--- Backups/Controller2/RAPID/TASK1/PROGMOD/CalibData.mod ---
MODULE CalibData
    PERS tooldata Tool_cow_catcher:=[TRUE,[[0,35.982,200],[1,0,0,0]],[1,[0,0,1],[1,0,0,0],0,0,0]];
    PERS tooldata Tool_Stack:=[TRUE,[[0,50,519.006],[1,0,0,0]],[1,[0,0,1],[1,0,0,0],0,0,0]];
    TASK PERS wobjdata wokOb_stak:=[FALSE,TRUE,"",[[1085.231623935,1226.713832798,-131.071212416],[0.707106781,0,0,-0.707106781]],[[0,0,0],[1,0,0,0]]];
    TASK PERS wobjdata WokOb_feed:=[FALSE,TRUE,"",[[1185.402623935,-706.018167202,-184.071212416],[0,1,0,0]],[[0,0,0],[1,0,0,0]]];
    TASK PERS wobjdata WokOb_feed1:=[FALSE,TRUE,"",[[1185.402623935,-706.018167202,-184.071212416],[0,1,0,0]],[[0,0,0],[1,0,0,0]]];
    TASK PERS wobjdata WokOb_Train_Top:=[FALSE,TRUE,"",[[58.90254417,-81.246884277,-27.346593322],[1,0.000000015,-0.00000002,-0.000000114]],[[-437.993,1154.838,527.576],[0,0,0.87019971,0.492699163]]];
    TASK PERS wobjdata WokOb_tarin_Front:=[FALSE,TRUE,"",[[58.90254417,-81.246884277,-27.346593322],[1,0.000000015,-0.00000002,-0.000000114]],[[-387.993,1035.72,66.547],[0.509717505,0.490089854,0.490089854,0.509717505]]];
    TASK PERS wobjdata Stand_tool_3:=[FALSE,TRUE,"",[[-537.392313736,-1111.43668764,-49.051212721],[0.707183689,0.000000377,0.000000377,-0.707029865]],[[0,0,0],[1,0,0,0]]];
    PERS tooldata Tooldata_2:=[TRUE,[[0,50,519.006],[1,0,0,0]],[1,[0,0,1],[1,0,0,0],0,0,0]];
    PERS tooldata Tooldata_3:=[TRUE,[[0,35.982,200],[1,0,0,0]],[1,[0,0,1],[1,0,0,0],0,0,0]];
    TASK PERS wobjdata WokOb_feed_1_Caw:=[FALSE,TRUE,"",[[1151.349623935,525.320832798,-184.071212416],[0,1,0,0]],[[0,0,0],[1,0,0,0]]];
    TASK PERS wobjdata WorOb_Stacl_Rb3:=[FALSE,TRUE,"",[[1166.594351677,998.920009045,-48.014532261],[0.705216396,-0.025578864,-0.025682184,-0.708064956]],[[0,0,0],[1,0,0,0]]];
ENDMODULE

--- Backups/Controller2/RAPID/TASK1/PROGMOD/Module1.mod ---
MODULE Module1
        CONST robtarget Target_10:=[[221.184118017,1602.844398512,1266.446017213],[0.128764321,-0.327741314,0.934862358,0.045141464],[-1,0,-1,0],[9E+09,9E+09,9E+09,9E+09,9E+09,9E+09]];
    CONST robtarget Target_20:=[[370.000026729,589.040405274,551.077515218],[0.04939984,-0.01732251,0.998628486,0.000856886],[-1,0,-1,0],[9E+09,9E+09,9E+09,9E+09,9E+09,9E+09]];
    CONST robtarget Target_30_up:=[[414.854817462,671.346228764,341.000522266],[0.000000533,0.00010877,0.999999994,0],[-1,0,0,0],[9E+09,9E+09,9E+09,9E+09,9E+09,9E+09]];
    CONST robtarget Target_30:=[[414.855137357,671.346228729,41.000522266],[0.000000533,0.00010877,0.999999994,0],[-1,0,0,0],[9E+09,9E+09,9E+09,9E+09,9E+09,9E+09]];
    CONST robtarget Target_40:=[[635.144122191,584.664958178,1616.637616509],[0.169784564,-0.794718952,0.515233089,0.27226798],[0,0,-1,0],[9E+09,9E+09,9E+09,9E+09,9E+09,9E+09]];
    CONST robtarget Target_50:=[[566.954133975,747.917817416,1065.318925343],[0.043909951,-0.83413114,0.542350178,0.090296418],[0,0,-1,0],[9E+09,9E+09,9E+09,9E+09,9E+09,9E+09]];
    CONST robtarget Target_60:=[[348.821647049,691.581522758,639.450946441],[0,-0.707106781,0.707106781,0],[0,0,0,0],[9E+09,9E+09,9E+09,9E+09,9E+09,9E+09]];
    CONST robtarget Target_70:=[[172.450821148,1938.736452761,-61.688697976],[0.659237738,-0.298307072,-0.108561129,-0.681639917],[1,0,-1,0],[9E+09,9E+09,9E+09,9E+09,9E+09,9E+09]];
    CONST robtarget Target_80:=[[569.616153696,1591.274414834,107.994145107],[0.624643546,-0.339078797,-0.046011146,-0.701946568],[1,-1,0,0],[9E+09,9E+09,9E+09,9E+09,9E+09,9E+09]];
    CONST robtarget Target_90:=[[387.500477242,662.643098431,-11.713507029],[0.624643546,-0.339078797,-0.046011146,-0.701946568],[1,0,-1,0],[9E+09,9E+09,9E+09,9E+09,9E+09,9E+09]];
    CONST robtarget Target_110:=[[166.316566086,558.37413423,-395.581097695],[0.714499458,0.106310973,-0.106526851,-0.683257295],[0,0,1,0],[9E+09,9E+09,9E+09,9E+09,9E+09,9E+09]];
    CONST robtarget Target_120:=[[-187.554461139,446.991796248,-213.907700592],[0.722131676,-0.014348091,0.019578353,-0.691329634],[0,0,1,0],[9E+09,9E+09,9E+09,9E+09,9E+09,9E+09]];
    CONST robtarget Target_140:=[[439.260504662,249.044211181,306.866921641],[0.012111654,0.04598783,0.712802443,-0.699750744],[1,-1,0,0],[9E+09,9E+09,9E+09,9E+09,9E+09,9E+09]];
    CONST robtarget Target_170:=[[536.884549621,570.585995165,-1132.877964218],[0.000000105,0.349155725,-0.000000008,0.937064715],[-1,0,-1,0],[9E+09,9E+09,9E+09,9E+09,9E+09,9E+09]];
    CONST robtarget Target_150:=[[205.16784185,570.586,-521.43503171],[-0.000000103,0.147809407,0.000000016,0.989015864],[0,-1,0,0],[9E+09,9E+09,9E+09,9E+09,9E+09,9E+09]];
    CONST robtarget Target_160:=[[178.331522758,542.515647049,-380.296079672],[0,0,0,1],[0,0,0,0],[9E+09,9E+09,9E+09,9E+09,9E+09,9E+09]];
    CONST robtarget Target_180:=[[416.962146713,864.683571188,1161.560654219],[0.40242565,-0.070024337,0.596108152,-0.691234591],[0,0,-1,0],[9E+09,9E+09,9E+09,9E+09,9E+09,9E+09]];
    CONST robtarget Target_190:=[[602.180688228,288.578411913,1239.026266106],[0.132681117,0.091945772,0.703686394,-0.691930022],[0,0,-1,0],[9E+09,9E+09,9E+09,9E+09,9E+09,9E+09]];
    CONST robtarget Target_Ro3_Cow_Pre_Last:=[[414.854817462,671.346228764,341.000522267],[0.000000533,0.00010877,0.999999994,0],[-1,0,0,0],[9E+09,9E+09,9E+09,9E+09,9E+09,9E+09]];
    CONST robtarget Target_Ro3_Cow_Last:=[[414.855137357,671.346228729,41.000522267],[0.000000533,0.00010877,0.999999994,0],[-1,0,0,0],[9E+09,9E+09,9E+09,9E+09,9E+09,9E+09]];
    CONST robtarget Target_R3_Caw_Pre_Last:=[[198.331522758,542.515647049,-580.296079672],[0.706823316,0.020019999,-0.020019999,-0.706823316],[-1,-1,0,0],[9E+09,9E+09,9E+09,9E+09,9E+09,9E+09]];
    CONST robtarget Target_200:=[[537.449802278,525.320832798,-1349.697350072],[0,0.093718973,0,0.995598691],[-1,0,-1,0],[9E+09,9E+09,9E+09,9E+09,9E+09,9E+09]];
    CONST robtarget Target_210:=[[395.399205293,525.320832798,-1001.535802608],[0.706823316,0.020019999,-0.020019999,-0.706823316],[-1,-1,0,0],[9E+09,9E+09,9E+09,9E+09,9E+09,9E+09]];
    CONST robtarget Target_R3_Caw_Last:=[[198.331522758,542.515647049,-380.296079672],[0.706823316,0.020019999,-0.020019999,-0.706823316],[-1,-1,0,0],[9E+09,9E+09,9E+09,9E+09,9E+09,9E+09]];
    CONST robtarget Target_R3_Caw_aT_Pre_Last:=[[602.180688228,308.563002126,1239.811220903],[0.132681117,0.091945772,0.703686394,-0.691930022],[0,0,-1,0],[9E+09,9E+09,9E+09,9E+09,9E+09,9E+09]];
    CONST robtarget Target_R3_Caw_aT_Last:=[[439.260504662,269.028801394,307.651876438],[0.009281573,0.046641452,0.754191684,-0.65493002],[0,0,-1,0],[9E+09,9E+09,9E+09,9E+09,9E+09,9E+09]];
    CONST robtarget Target_230:=[[431.630872596,635.901601801,1236.076927583],[0.024057172,-0.814914042,0.571422358,0.093876759],[0,0,-1,0],[9E+09,9E+09,9E+09,9E+09,9E+09,9E+09]];
    CONST robtarget Target_Ro3_Stack_Pre_last:=[[242.865175793,579.269518535,748.277875669],[0.025682184,0.708064956,-0.705216396,-0.025578864],[0,0,0,0],[9E+09,9E+09,9E+09,9E+09,9E+09,9E+09]];
    CONST robtarget Target_Ro3_Stack_last:=[[228.375978011,579.211110467,548.803416812],[0.025682184,0.708064956,-0.705216396,-0.025578864],[0,0,0,0],[9E+09,9E+09,9E+09,9E+09,9E+09,9E+09]];
    CONST robtarget Target_220:=[[578.676966526,497.743647902,1659.839754198],[0.150831029,-0.765727927,0.566419369,0.264725973],[0,0,-1,0],[9E+09,9E+09,9E+09,9E+09,9E+09,9E+09]];
    CONST robtarget Target_240:=[[49.842979194,487.554033752,-1340.183033329],[0.336292984,-0.171245379,-0.062328221,-0.923957381],[-1,0,-1,0],[9E+09,9E+09,9E+09,9E+09,9E+09,9E+09]];
    CONST robtarget Target_250:=[[283.995850065,381.102635573,-1044.400341171],[0.707106781,0,0,-0.707106781],[-1,-1,1,0],[9E+09,9E+09,9E+09,9E+09,9E+09,9E+09]];
    CONST robtarget Target_Rb3_Stack_Pre_Last:=[[270.393522758,498.685647049,-819.068079672],[0.707106781,0,0,-0.707106781],[-1,0,0,0],[9E+09,9E+09,9E+09,9E+09,9E+09,9E+09]];
    CONST robtarget Target_Rb3_Stack_Last:=[[270.393522758,498.685647049,-299.068079672],[0.707106781,0,0,-0.707106781],[-1,0,0,0],[9E+09,9E+09,9E+09,9E+09,9E+09,9E+09]];
    CONST robtarget Target_Stack_2_Pre:=[[168.638525927,1312.987191107,-158.731374197],[0.924786368,-0.310928816,0.214202621,-0.047017889],[1,1,-2,0],[9E+09,9E+09,9E+09,9E+09,9E+09,9E+09]];
    CONST robtarget Target_Stack_4_last:=[[389.005720296,705.812701337,80.121150632],[0.961548171,-0.165322925,0.204449569,-0.07933359],[1,-1,0,0],[9E+09,9E+09,9E+09,9E+09,9E+09,9E+09]];
    CONST robtarget Target_Stack_3_Pre_last:=[[389.005720296,877.311368754,-22.777863329],[0.623819913,-0.261468638,0.027666715,-0.736014552],[1,-1,0,0],[9E+09,9E+09,9E+09,9E+09,9E+09,9E+09]];
    CONST robtarget Target_Stack_1_Start:=[[-788.497531681,1603.313448753,-159.059404418],[0.940109898,-0.316080846,-0.12465014,0.027360947],[0,1,-1,0],[9E+09,9E+09,9E+09,9E+09,9E+09,9E+09]];
    CONST robtarget Target_Stack_3_last:=[[389.005720296,963.060702463,-74.227370309],[0.961548171,-0.165322925,0.204449569,-0.07933359],[1,-1,0,0],[9E+09,9E+09,9E+09,9E+09,9E+09,9E+09]];
    CONST robtarget Target_270:=[[381.16653399,952.850551141,-196.906188778],[0.952856429,-0.264493422,0.136128666,-0.059806695],[1,0,-1,0],[9E+09,9E+09,9E+09,9E+09,9E+09,9E+09]];
    CONST robtarget Target_270_2:=[[381.16652599,1124.349221645,-299.805197594],[0.952856429,-0.264493422,0.136128666,-0.059806695],[1,1,-1,0],[9E+09,9E+09,9E+09,9E+09,9E+09,9E+09]];
!***********************************************************
    !
    ! Module:  Module1
    !
    ! Description:
    !   <Insert description here>
    !
    ! Author: haba0028
    !
    ! Version: 1.0
    !
    !***********************************************************


    !***********************************************************
    !
    ! Procedure main
    !
    !   This is the entry point of your program
    !
    !***********************************************************
    PROC main()
        !Add your code here
        SetDo doAt_Tool_SC1,0;
        SetDO doGrepCaw,0;
        SetDo doGrepStak,0;
        WaitDI di_Atctive,1;





        Path_Att_tool_cow;
        Path_Att_cow_tR;
        Path_Att_cow_tT;
        Path_diAtt_tool_cow;


        Path_Rob3_att_tool_stak;
        Path_Rb3_Att_Stack_tR;
        Path_Rob3_att_tT_Stack;
        Path_Rob3_diatt_tool_stak;



!        Path_Rob3_att_tT_Stack;
    ENDPROC

    PROC Path_Att_tool_cow()
        MoveJ Target_10,v1000,fine,tool0\WObj:=Stand_tool_3;
        MoveL Target_20,v1000,fine,tool0\WObj:=Stand_tool_3;
        MoveL Target_Ro3_Cow_Pre_Last,v1000,fine,tool0\WObj:=Stand_tool_3;
        MoveL Target_Ro3_Cow_Last,v1000,fine,tool0\WObj:=Stand_tool_3;
        WaitTime 0.3;
        SetDo doAt_Tool_SC1,1;
        WaitTime 1;
        MoveL Target_Ro3_Cow_Pre_Last,v1000,fine,Tool_cow_catcher\WObj:=Stand_tool_3;
        MoveL Target_20,v1000,fine,Tool_cow_catcher\WObj:=Stand_tool_3;
        MoveL Target_10,v1000,fine,Tool_cow_catcher\WObj:=Stand_tool_3;
    ENDPROC
    PROC Path_diAtt_tool_cow()
        WaitTime 0.3;
        MoveJ Target_10,v1000,fine,Tool_cow_catcher\WObj:=Stand_tool_3;
        MoveL Target_20,v1000,fine,Tool_cow_catcher\WObj:=Stand_tool_3;
        MoveL Target_Ro3_Cow_Pre_Last,v1000,fine,Tool_cow_catcher\WObj:=Stand_tool_3;
        MoveL Target_Ro3_Cow_Last,v1000,fine,tool0\WObj:=Stand_tool_3;
        WaitTime 0.3;
        SetDo doAt_Tool_SC1,0;
        WaitTime 1;
        MoveL Target_Ro3_Cow_Pre_Last,v1000,fine,tool0\WObj:=Stand_tool_3;
        MoveL Target_20,v1000,fine,tool0\WObj:=Stand_tool_3;
        MoveL Target_10,v1000,fine,tool0\WObj:=Stand_tool_3;
    ENDPROC

    PROC Path_Rob3_att_tool_stak()
        MoveJ Target_220,v1000,fine,tool0\WObj:=WorOb_Stacl_Rb3;
        MoveL Target_230,v1000,fine,tool0\WObj:=WorOb_Stacl_Rb3;
        MoveL Target_Ro3_Stack_Pre_last,v1000,fine,tool0\WObj:=WorOb_Stacl_Rb3;
        MoveL Target_Ro3_Stack_last,v1000,fine,tool0\WObj:=WorOb_Stacl_Rb3;
        WaitTime 0.3;
        SetDo doAt_Tool_SC1,1;
        WaitTime 1;
        MoveL Target_Ro3_Stack_Pre_last,v1000,fine,Tool_Stack\WObj:=WorOb_Stacl_Rb3;
        MoveL Target_230,v1000,fine,Tool_Stack\WObj:=WorOb_Stacl_Rb3;
        MoveL Target_220,v1000,fine,Tool_Stack\WObj:=WorOb_Stacl_Rb3;
    ENDPROC

    PROC Path_Rob3_diatt_tool_stak()
        MoveJ Target_220,v1000,fine,Tool_Stack\WObj:=WorOb_Stacl_Rb3;
        MoveL Target_230,v1000,fine,Tool_Stack\WObj:=WorOb_Stacl_Rb3;
        MoveL Target_Ro3_Stack_Pre_last,v1000,fine,Tool_Stack\WObj:=WorOb_Stacl_Rb3;
        MoveL Target_Ro3_Stack_last,v1000,fine,tool0\WObj:=WorOb_Stacl_Rb3;
        WaitTime 0.3;
        SetDo doAt_Tool_SC1,0;
        WaitTime 1;
        MoveL Target_Ro3_Stack_Pre_last,v1000,fine,tool0\WObj:=WorOb_Stacl_Rb3;
        MoveL Target_230,v1000,fine,tool0\WObj:=WorOb_Stacl_Rb3;
        MoveL Target_220,v1000,fine,tool0\WObj:=WorOb_Stacl_Rb3;
    ENDPROC







    PROC Path_Att_cow_tR()
        WaitTime 0.3;
        MoveJ Target_200,v1000,fine,Tool_cow_catcher\WObj:=WokOb_feed_1_Caw;
        MoveL Target_210,v1000,fine,Tool_cow_catcher\WObj:=WokOb_feed_1_Caw;
        MoveL Target_R3_Caw_Pre_Last,v1000,fine,Tool_cow_catcher\WObj:=WokOb_feed_1_Caw;
        MoveL Target_R3_Caw_Last,v1000,fine,Tool_cow_catcher\WObj:=WokOb_feed_1_Caw;
        WaitTime 0.3;
        SetDO doGrepCaw,1;
        WaitTime 1;
        MoveL Target_R3_Caw_Pre_Last,v1000,fine,Tool_cow_catcher\WObj:=WokOb_feed_1_Caw;
        MoveL Target_210,v1000,fine,Tool_cow_catcher\WObj:=WokOb_feed_1_Caw;
        MoveL Target_200,v1000,fine,Tool_cow_catcher\WObj:=WokOb_feed_1_Caw;
    ENDPROC

    PROC Path_Rb3_Att_Stack_tR()
        WaitTime 0.3;
        MoveJ Target_240,v1000,fine,Tool_Stack\WObj:=WokOb_feed;
        MoveL Target_250,v1000,fine,Tool_Stack\WObj:=WokOb_feed;
        MoveL Target_Rb3_Stack_Pre_Last,v1000,fine,Tool_Stack\WObj:=WokOb_feed;
        MoveL Target_Rb3_Stack_Last,v1000,fine,Tool_Stack\WObj:=WokOb_feed;
        WaitTime 0.3;
        SetDo doGrepStak,1;
        WaitTime 1;
        MoveL Target_Rb3_Stack_Pre_Last,v1000,fine,Tool_Stack\WObj:=WokOb_feed;
        MoveL Target_250,v1000,fine,Tool_Stack\WObj:=WokOb_feed;
        MoveL Target_240,v1000,fine,Tool_Stack\WObj:=WokOb_feed;
    ENDPROC


    PROC Path_Att_cow_tT()
        WaitTime 0.3;
        MoveJ Target_180,v1000,fine,Tool_cow_catcher\WObj:=WokOb_tarin_Front;
        MoveL Target_R3_Caw_aT_Pre_Last,v1000,fine,Tool_cow_catcher\WObj:=WokOb_tarin_Front;
        MoveL Target_R3_Caw_aT_Last,v1000,fine,Tool_cow_catcher\WObj:=WokOb_tarin_Front;
        WaitTime 0.3;
        SetDO doGrepCaw,0;
        WaitTime 1;
        MoveL Target_R3_Caw_aT_Pre_Last,v1000,fine,tool0\WObj:=WokOb_tarin_Front;
        MoveL Target_180,v1000,fine,tool0\WObj:=WokOb_tarin_Front;
    ENDPROC

    PROC Path_Rob3_att_tT_Stack()
        WaitTime 0.3;
        MoveJ Target_Stack_1_Start,v1000,fine,Tool_Stack\WObj:=WokOb_Train_Top;
        MoveL Target_270_2,v1000,fine,Tool_Stack\WObj:=WokOb_Train_Top;
        MoveL Target_270,v1000,fine,Tool_Stack\WObj:=WokOb_Train_Top;
        WaitTime 0.3;
        SetDo doGrepStak,0;
        WaitTime 1;
        MoveL Target_270_2,v1000,fine,Tool_Stack\WObj:=WokOb_Train_Top;
        MoveL Target_Stack_1_Start,v1000,fine,Tool_Stack\WObj:=WokOb_Train_Top;
    ENDPROC

ENDMODULE

--- Backups/Controller1/SYSPAR/EIO.cfg ---
EIO:CFG_1.0:6:1::
#
INDUSTRIAL_NETWORK:

      -Name "PROFIBUS" -Label "PROFIBUS Controller Network"\
      -CfgPath "HOME/pbus_cfg.bin"
#
PROFIBUS_DEVICE:

      -Name "Board10"
#
EIO_SIGNAL:

      -Name "diAttachTool" -SignalType "DO" -Device "Board10" -DeviceMap "0"

      -Name "doAttachTool" -SignalType "DO" -Device "Board10" -DeviceMap "1"

      -Name "doAttachTo_S" -SignalType "DO" -Device "Board10" -DeviceMap "2"

      -Name "doAtWhRi" -SignalType "DO" -Device "Board10" -DeviceMap "3"

      -Name "Att_link" -SignalType "DO" -Device "Board10" -DeviceMap "4"

      -Name "doAT_Left" -SignalType "DO" -Device "Board10" -DeviceMap "5"

      -Name "doAt_Wh_Left" -SignalType "DO" -Device "Board10" -DeviceMap "6"

      -Name "doAt_Link_Left" -SignalType "DO" -Device "Board10" -DeviceMap "7"

      -Name "doAt_AxelP_Left" -SignalType "DO" -Device "Board10" -DeviceMap "8"

      -Name "doAt_Arm_Left" -SignalType "DO" -Device "Board10" -DeviceMap "9"

      -Name "doAt_AxelP_Right" -SignalType "DO" -Device "Board10"\
      -DeviceMap "10"

      -Name "doAt_ArmP_Right" -SignalType "DO" -Device "Board10" -DeviceMap "11"

--- Backups/Controller2/SYSPAR/EIO.cfg ---
EIO:CFG_1.0:6:1::
#
INDUSTRIAL_NETWORK:

      -Name "PROFIBUS" -Label "PROFIBUS Controller Network"\
      -CfgPath "HOME/pbus_cfg.bin"
#
PROFIBUS_DEVICE:

      -Name "Board20"
#
EIO_SIGNAL:

      -Name "di_Atctive" -SignalType "DI" -Device "Board20" -DeviceMap "0"

      -Name "doAt_Tool_SC1" -SignalType "DO" -Device "Board20" -DeviceMap "1"

      -Name "doGrepCaw" -SignalType "DO" -Device "Board20" -DeviceMap "2"

      -Name "doGrepStak" -SignalType "DO" -Device "Board20" -DeviceMap "3"
